TYPE ST_Softsettings_AcDcCharger :
STRUCT
	b_Enable 			: BOOL;
	r_CurrentSetpoint	: REAL;
	r_PowerSetpoint 	: REAL;
	r_SocTarget			: REAL;
	r_MinACVoltage		: REAL;
	e_ControlType		: ePowerControlType := ePowerControlType.Current;
END_STRUCT
END_TYPE

(* stored: Version 1.1.0.1, ProductVersion 3.1.4026.18
   DUT ST_Softsettings_AcDcCharger: Id {982a6180-2592-4114-b44b-7b43e0165286} *)
